{attribute addProperty BoxType "EL3602-0002-0016"}
{attribute addProperty Id "StatusAT %I*Status_C6F82E6F1621ValueAT %I*DINT32417"}
{attribute addProperty CRC "3201558924"}
{attribute addProperty SizeInBites "48"}
{attribute addProperty SizeInBytes "6"}
TYPE AI_Inputs_Channel_BED3E98C :
STRUCT
	{attribute addProperty Name "Status"}
	Status AT %I* : Status_C6F82E6F;
	{attribute addProperty Name "Value"}
	Value AT %I* : DINT;
END_STRUCT
END_TYPE

(* stored: Version 1.2.0.0, ProductVersion 3.1.4024.9
   DUT AI_Inputs_Channel_BED3E98C: Id {c97e564f-3d44-4654-92c8-0569e308fd3e} *)
